// TIA Portal V17 export
// export: Created 2024-09-02T12:50:40.8865723Z, ExportSetting WithDefaults, DisplayName Totally Integrated Automation Portal, DisplayVersion V17, DisplayName TIA Portal Openness, DisplayVersion V17, DisplayName TIA Portal Version Control Interface, DisplayVersion V17, DisplayName STEP 7 Professional, DisplayVersion V17, DisplayName STEP 7 Safety, DisplayVersion V17, DisplayName WinCC Professional, DisplayVersion V17
TYPE "Aveva_Result_Global_Result_Station"
// stored: IsFailsafeCompliant false
   STRUCT
      Station_Status { ExternalWritable := 'False'} : Struct
         Started { ExternalWritable := 'False'} : Bool;   // Work Started
         Finished_NOK { ExternalWritable := 'False'} : Bool;   // Work Finished NOK
         Finished_OK { ExternalWritable := 'False'} : Bool;   // Work Finished OK
         Bypassed { ExternalWritable := 'False'} : Bool;   // Work Bypassed
         Interrupted { ExternalWritable := 'False'} : Bool;   // Work Interrupted
      END_STRUCT;
   END_STRUCT;
END_TYPE
